{attribute 'linkalways'} 
{attribute 'no_explicit_call' := 'This FB is a CLASS and must be accessed using methods or properties'}
{attribute 'enable_dynamic_creation'}
FUNCTION_BLOCK FINAL MIN_ULINT EXTENDS Node
VAR
	in1 : _ULINT(0);
	in2 : _ULINT(0);
	out : _ULINT(0);
END_VAR

METHOD PUBLIC Clone : I_Node
VAR
	pNode : POINTER TO MIN_ULINT;
END_VAR
pNode := __NEW(MIN_ULINT);
Clone := pNode^;
END_METHOD

METHOD FB_init : BOOL
VAR_INPUT
	bInitRetains : BOOL; // if TRUE, the retain variables are initialized (warm start / cold start)
	bInCopyCode : BOOL;  // if TRUE, the instance afterwards gets moved into the copy code (online change)
END_VAR
AddInput('in1',THIS^.in1);
AddInput('in2',THIS^.in2);
AddOutput('out', THIS^.out);
END_METHOD

METHOD PROTECTED OnExecute
VAR
END_VAR
out.Value := MIN(in1.Value, in2.Value);
END_METHOD

END_FUNCTION_BLOCK

(* stored: Version 1.1.0.1, ProductVersion 3.1.4024.15
   POU MIN_ULINT: Id {09107673-8590-4bc3-bbd1-aebdbaf6e698}, SpecialFunc None
   Folder Constructor: Id {6d968a74-84ad-43f9-b754-d7ad4e74ed5d}
   Method Clone: Id {59d41dcb-5433-4444-8139-40227c276068}
   Method FB_init: Id {8057afb6-11c4-4f4e-ae8e-7ece2c90210c}
   Method OnExecute: Id {13f3c6a8-c471-47a9-97e0-a7efd873ae1a} *)
